// TIA Portal V16 export
// export: Created 2021-08-10T09:04:59.8060586Z, ExportSetting WithDefaults, WithReadOnly, DisplayName Totally Integrated Automation Portal, DisplayVersion V16, DisplayName TIA Portal Version Control Interface, DisplayVersion V16, DisplayName TIA Portal Openness, DisplayVersion V16, DisplayName TIA Portal Teamcenter Gateway, DisplayVersion V16, DisplayName SINAMICS Startdrive Advanced, DisplayVersion V16, DisplayName SINAMICS Startdrive G130, G150, S120, S150, SINAMICS MV, S210, DisplayVersion V16, DisplayName SINAMICS Startdrive G110M, G120, G120C, G120D, G120P, DisplayVersion V16, DisplayName STEP 7 Professional, DisplayVersion V16, DisplayName STEP 7 Safety, DisplayVersion V16, DisplayName WinCC Unified SCADA Engineering System, DisplayVersion V16
DATA_BLOCK "DB_ProgramLogic"   // DB4
{ S7_Optimized_Access := 'TRUE' }
VERSION : 0.1
// stored: AutoNumber true, CodeModifiedDate 2020-02-26T07:40:10.2847553Z, CompileDate 2021-07-03T08:38:37.7718266Z, CreationDate 2020-02-26T07:39:28.2364137Z, DBAccessibleFromOPCUA true, DownloadWithoutReinit false, InterfaceModifiedDate 2020-02-26T07:40:10.2847553Z, IsConsistent true, IsKnowHowProtected false, IsOnlyStoredInLoadMemory false, IsPLCDB false, IsRetainMemResEnabled false, IsWriteProtectedInAS false, MemoryReserve 100, ModifiedDate 2020-02-26T07:40:10.2847553Z, ParameterModified 2020-02-26T07:40:10.2847553Z, StructureModified 2020-02-26T07:40:10.2847553Z
   VAR
      VlvLiq1_Open : Bool;
      VlvLiq2_Open : Bool;
      VlvDrn_Open : Bool;
   END_VAR
BEGIN
END_DATA_BLOCK
